# B&R Automation Studio project Test_Version_Control
Automation Studio 4.9

## Configuration Config1

### Hardware
```
X20CP1586 : X20CP1586 v1.10.0.0
  Connector IF2:
    ActivateDevice = 1
  ConfigurationID = Test01_Version_Control_Config1
  FileDevice1
  FileDeviceName1 = USER
  FileDevicePath1 = USER_PATH
```

## Logical view

### Global.var - Global variables
```iecst
VAR
	BtnStart : BOOL;
	BtnStop : BOOL;
	BtnEmStop : BOOL;
	MotorConveyorFwd : BOOL;
	MotorConveyorRev : BOOL;
//This command Tests the connection of Jira to GitHub
	RobotCodeJira : BOOL;
//This command Tests the connection of Jira to GitHub
	RobotCodeJira : BOOL;
//This command Tests the connection of Jira to GitHub
	RobotCodeJira : BOOL;
END_VAR
```

### Program Logical/Program (IEC)

#### Main.st
```iecst
PROGRAM _INIT
	(* Insert code here *)

	//BtnStart : BOOL;
//	BtnStop : BOOL;
	//MotorConveyor : BOOL;

END_PROGRAM

PROGRAM _CYCLIC
	(* Insert code here *)

	IF BtnStart THEN
		MotorConveyor := TRUE;
	ELSIF BtnStop THEN
		MotorConveyor := FALSE;
	END_IF

END_PROGRAM

PROGRAM _EXIT
	(* Insert code here *)
	IF BtnStop THEN
	MotorConveyor := FALSE;
	END_IF

END_PROGRAM
```

Listed in the project but not available here: Logical/Global.typ, Logical/Libraries, Logical/TS_UnitTest
